INTERFACE ITcoComponent EXTENDS ITcoObject,ITcoRestorable

METHOD PUBLIC Maintenance
END_METHOD

END_INTERFACE

(* stored: Version 1.1.0.1, ProductVersion 3.1.4024.6
   Itf ITcoComponent: Id {226fd2d6-401e-4c29-97f4-f7e58b55d445}
   Method Maintenance: Id {b2fe216f-37ab-46ad-9d62-c3f8870418e6} *)
